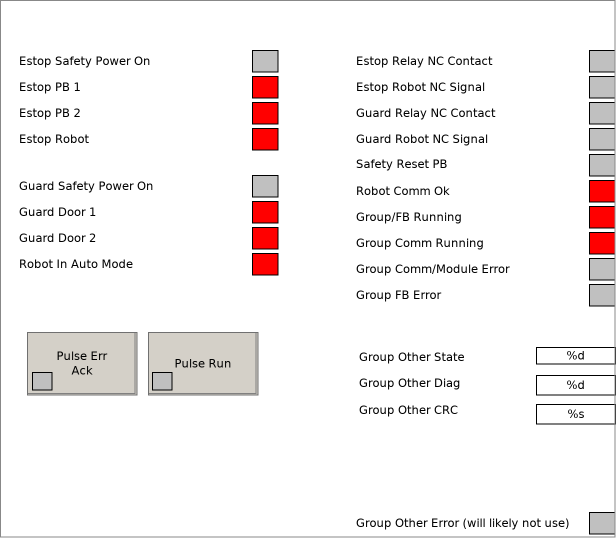
VISUALIZATION Safety  // 616x538
    Rectangle (252,50 26x22), colour toggle: Stn054_03_SafetyInterface.hoSafetyPowerOn_Estop
    Rectangle (16,46 224x30), "Estop Safety Power On"
    Rectangle (252,76 26x22), colour toggle: Stn054_03_SafetyInterface.hoEstopPB1Ok
    Rectangle (16,72 224x30), "Estop PB 1"
    Rectangle (252,102 26x22), colour toggle: Stn054_03_SafetyInterface.hoEstopPB2Ok
    Rectangle (16,98 224x30), "Estop PB 2"
    Rectangle (252,128 26x22), colour toggle: Stn054_03_SafetyInterface.hoEstopRobotOk
    Rectangle (16,124 224x30), "Estop Robot"
    Rectangle (252,175 26x22), colour toggle: Stn054_03_SafetyInterface.hoSafetyPowerOn_Guard
    Rectangle (16,171 224x30), "Guard Safety Power On"
    Rectangle (252,201 26x22), colour toggle: Stn054_03_SafetyInterface.hoGuardDoor1Ok
    Rectangle (16,197 224x30), "Guard Door 1"
    Rectangle (252,227 26x22), colour toggle: Stn054_03_SafetyInterface.hoGuardDoor2Ok
    Rectangle (16,223 224x30), "Guard Door 2"
    Rectangle (252,253 26x22), colour toggle: Stn054_03_SafetyInterface.hoRobotInAutoMode
    Rectangle (16,249 224x30), "Robot In Auto Mode"
    Rectangle (589,50 26x22), colour toggle: Stn054_03_SafetyInterface.hoRelayNCContact_Estop
    Rectangle (353,46 224x30), "Estop Relay NC Contact"
    Rectangle (589,76 26x22), colour toggle: Stn054_03_SafetyInterface.hoRobotNCContact_Estop
    Rectangle (353,72 224x30), "Estop Robot NC Signal"
    Rectangle (589,102 26x22), colour toggle: Stn054_03_SafetyInterface.hoRelayNCContact_Guard
    Rectangle (353,98 224x30), "Guard Relay NC Contact"
    Rectangle (589,128 26x22), colour toggle: Stn054_03_SafetyInterface.hoRobotNCContact_Guard
    Rectangle (353,124 224x30), "Guard Robot NC Signal"
    Rectangle (589,180 26x22), colour toggle: Stn054_03_SafetyInterface.hoRobotCommOk
    Rectangle (353,176 224x30), "Robot Comm Ok"
    Rectangle (589,206 26x22), colour toggle: Stn054_03_SafetyInterface.hoSafetyGroupAndFBInRun
    Rectangle (353,202 224x30), "Group/FB Running"
    Rectangle (589,232 26x22), colour toggle: Stn054_03_SafetyInterface.hoSafetyGroupComRunning
    Rectangle (353,228 224x30), "Group Comm Running"
    Rectangle (589,258 26x22), colour toggle: Stn054_03_SafetyInterface.hoSafetyGroupComErr
    Rectangle (353,254 224x30), "Group Comm/Module Error"
    Rectangle (589,284 26x22), colour toggle: Stn054_03_SafetyInterface.hoSafetyGroupFBErr
    Rectangle (353,280 224x30), "Group FB Error"
    Rectangle (589,512 26x22), colour toggle: Stn054_03_SafetyInterface.hoSafetyGroupOtherErr
    Rectangle (353,508 224x30), "Group Other Error (will likely not use)"
    Rectangle (356,342 224x30), "Group Other State"
    Rectangle (356,368 224x30), "Group Other Diag"
    Rectangle (536,347 80x17), "%d", text variable: Stn054_03_SafetyInterface.hoSafetyGroup_State
    Rectangle (536,375 80x20), "%d", text variable: Stn054_03_SafetyInterface.hoSafetyGroup_Diag
    Button (27,332 110x63), "Pulse Err Ack"
        tap Stn054_03_SafetyInterface.hiSafetyGroupPulseErrAck
    Button (148,332 110x63), "Pulse Run"
        tap Stn054_03_SafetyInterface.hiSafetyGroupPulseRun
    Rectangle (152,372 20x18), colour toggle: Stn054_03_SafetyInterface.hoSafetyGroupRun
    Rectangle (32,372 20x18), colour toggle: Stn054_03_SafetyInterface.hoSafetyGroupErrAck
    Rectangle (356,395 224x30), "Group Other CRC"
    RoundedRectangle (536,404 80x20), "%s", text variable: Stn054_03_SafetyInterface.hoSafetyCtrlCRC, colour variable: 16#FF000000 OR (16#FF000000 OR (Global_Variables.gStn100.OperatorMessage.Color))
    Rectangle (589,154 26x22), colour toggle: Stn054_03_SafetyInterface.hoSafetyResetPB
    Rectangle (353,149 224x30), "Safety Reset PB"
END_VISUALIZATION

(* stored: Version 1.1.0.1, ProductVersion 3.1.4024.6
   Visu Safety: Id {d0f26792-cb29-4b70-8770-1744df3526ef} *)
